FUNCTION_BLOCK FB_EventBuffer
VAR
    MemRingBuffer : FB_MemRingBuffer;
	BufferArray : ARRAY[0..MAX_BUFFER_SIZE] OF BYTE;
END_VAR
VAR CONSTANT
	SIZE_OF_ST_EVENT : UDINT := SIZEOF(ST_Event);
	MAX_NUMBER_OF_ST_EVENTS : UDINT := 5;
	MAX_BUFFER_SIZE : UDINT := SIZE_OF_ST_EVENT * MAX_NUMBER_OF_ST_EVENTS + SIZEOF(MemRingBuffer);
END_VAR

METHOD PUBLIC AddEvent
VAR_INPUT
	stEvent : REFERENCE TO ST_Event;
END_VAR
VAR_OUTPUT
	bError : BOOL;
END_VAR
MemRingBuffer.A_AddTail(pWrite := ADR(stEvent), 
						cbWrite := SIZEOF(stEvent), 
						pBuffer := ADR(BufferArray), 
						cbBuffer := SIZEOF(BufferArray));
						
bError := NOT MemRingBuffer.bOk;
END_METHOD

METHOD PUBLIC GetAndRemoveEvent
VAR_OUTPUT
	stEvent : ST_Event;
	bError : BOOL;
END_VAR
MemRingBuffer.A_RemoveHead(pRead := ADR(stEvent), cbRead := SIZEOF(stEvent), pBuffer := ADR(BufferArray), cbBuffer := SIZEOF(BufferArray));
						
bError := NOT MemRingBuffer.bOk;
END_METHOD

END_FUNCTION_BLOCK

(* stored: Version 1.1.0.1, ProductVersion 3.1.4024.12
   POU FB_EventBuffer: Id {376bb73c-8cf7-4495-bc60-f00000825dae}, SpecialFunc None
   Method AddEvent: Id {9ae709c7-2660-4275-8f01-69159fe1f889}
   Method GetAndRemoveEvent: Id {2057184e-7bd0-4432-9336-243d9737a077} *)
